TYPE ZComUnit :
STRUCT
{region "Picker"}
{IF NOT (defined (Picker_disabled))}
  Picker : PickerCom;
  {attribute 'ZId' := 'c43c28b7-9e8c-48c6-a4f8-946be27888d3'}
{END_IF}
{endregion}
{attribute '__ZwPlcApplicationComUnitDeclaration__'} // Do not remove this attribute! It is used for code generation.
END_STRUCT
END_TYPE

(* stored: Version 1.1.0.1
   DUT ZComUnit: Id {dcdd230e-27a3-485c-b060-79109a96f888} *)
